// Gets the upper bound index of the array of specified type.
FUNCTION F_GetDateAndTimeArrayUpperBound : T_Position // The upper bound index of the specified array.
VAR_IN_OUT
	arArray : ARRAY[*] OF DATE_AND_TIME; // The array to query.
END_VAR

F_GetDateAndTimeArrayUpperBound := UPPER_BOUND(arArray, 1);

END_FUNCTION

(* stored: Version 1.1.0.1
   POU F_GetDateAndTimeArrayUpperBound: Id {48dc808f-54de-02e6-1c0f-d3b75341756b}, SpecialFunc None *)
